// Mitsubishi GX Works2 project: plc_q1   PLC: FX1N/FX1NC

PROGRAM MAIN
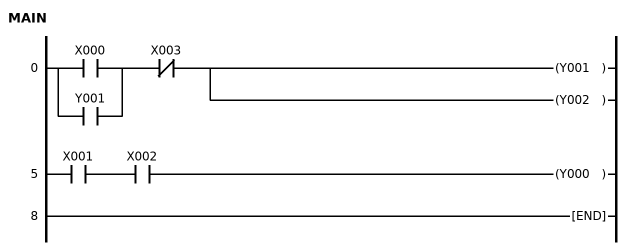
0     LD      X000
      OR      Y001
      ANI     X003
      OUT     Y001
      OUT     Y002
5     LD      X001
      AND     X002
      OUT     Y000
8     END
END_PROGRAM
